FUNCTION_BLOCK M3IO EXTENDS SM_M3IO
VAR_INPUT
END_VAR
VAR_OUTPUT
END_VAR
VAR
    _testVar : INT;
END_VAR

SUPER^();

// do stuff

//SUPER^();

END_FUNCTION_BLOCK

(* stored: Version 1.1.0.1, ProductVersion 3.1.4018.2
   POU M3IO: Id {d2eb1c04-ac54-45c4-9062-d9fdf96add18}, SpecialFunc None *)
